# EPICS substitutions: iocBoot/iocAMControls/amcontrols.substitutions
file "$(TOP)/db/amControls.template"
{
pattern
{  P,      R,     }
{32id:, AMControls:, }
}
